% RSLogix 500 project High Pressure Washer no labels Veracruz.RSS, saved by version 11.00.00.00 %
PROJECT "UNTITLED"    % processor: MicroLogix 1400 %

PROGRAM FILES
  LAD 2   7 rungs
  LAD 3   25 rungs
  LAD 4   18 rungs
  LAD 5   20 rungs
  LAD 6   10 rungs
  LAD 7   39 rungs
  LAD 8   15 rungs
  LAD 9, 10, 11, 12, 13, 14, 15: only END

DATA FILES
  O0 OUTPUT  10 elements
  I1 INPUT  17 elements
  S2 STATUS  66 elements
  B3 BINARY  32 elements
  T4 TIMER  40 elements
  C5 COUNTER  32 elements
  R6 CONTROL  16 elements
  N7 INTEGER  110 elements
  F8 RESERVED  1 elements
  PD9   4 elements

LADDER 2
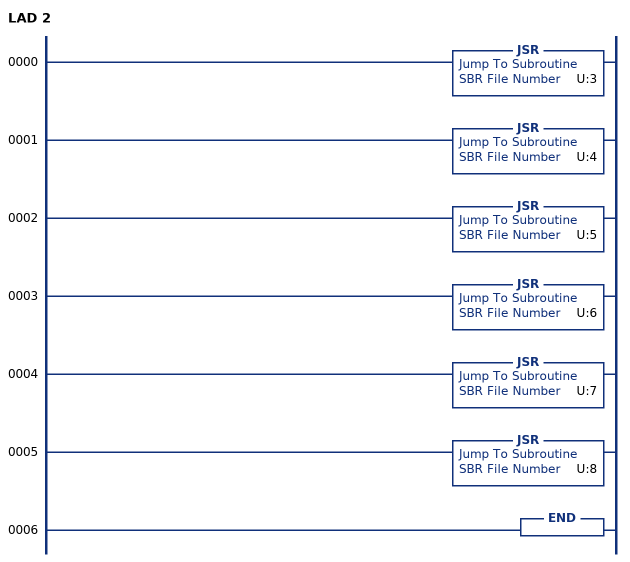
% Rung: 0 %
SOR JSR U:3 EOR
% Rung: 1 %
SOR JSR U:4 EOR
% Rung: 2 %
SOR JSR U:5 EOR
% Rung: 3 %
SOR JSR U:6 EOR
% Rung: 4 %
SOR JSR U:7 EOR
% Rung: 5 %
SOR JSR U:8 EOR
% Rung: 6 %
SOR END EOR

LADDER 3
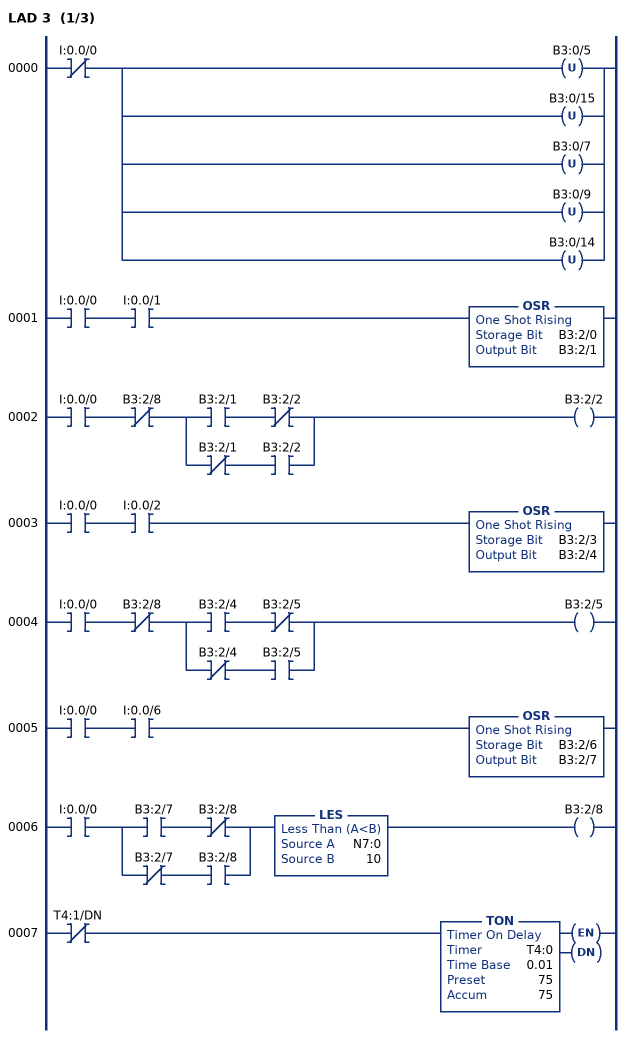
% Rung: 0 %
SOR XIO I:0.0/0 BST BST BST BST OTU B3:0/5 NXB OTU B3:0/15 BND NXB OTU B3:0/7 BND NXB OTU B3:0/9 BND NXB OTU B3:0/14 BND EOR
% Rung: 1 %
SOR XIC I:0.0/0 XIC I:0.0/1 OSR B3:2/0 B3:2/1 EOR
% Rung: 2 %
SOR XIC I:0.0/0 XIO B3:2/8 BST XIC B3:2/1 XIO B3:2/2 NXB XIO B3:2/1 XIC B3:2/2 BND OTE B3:2/2 EOR
% Rung: 3 %
SOR XIC I:0.0/0 XIC I:0.0/2 OSR B3:2/3 B3:2/4 EOR
% Rung: 4 %
SOR XIC I:0.0/0 XIO B3:2/8 BST XIC B3:2/4 XIO B3:2/5 NXB XIO B3:2/4 XIC B3:2/5 BND OTE B3:2/5 EOR
% Rung: 5 %
SOR XIC I:0.0/0 XIC I:0.0/6 OSR B3:2/6 B3:2/7 EOR
% Rung: 6 %
SOR XIC I:0.0/0 BST XIC B3:2/7 XIO B3:2/8 NXB XIO B3:2/7 XIC B3:2/8 BND LES N7:0 10 OTE B3:2/8 EOR
% Rung: 7 %
SOR XIO T4:1/DN TON T4:0 0.01 75 75 EOR

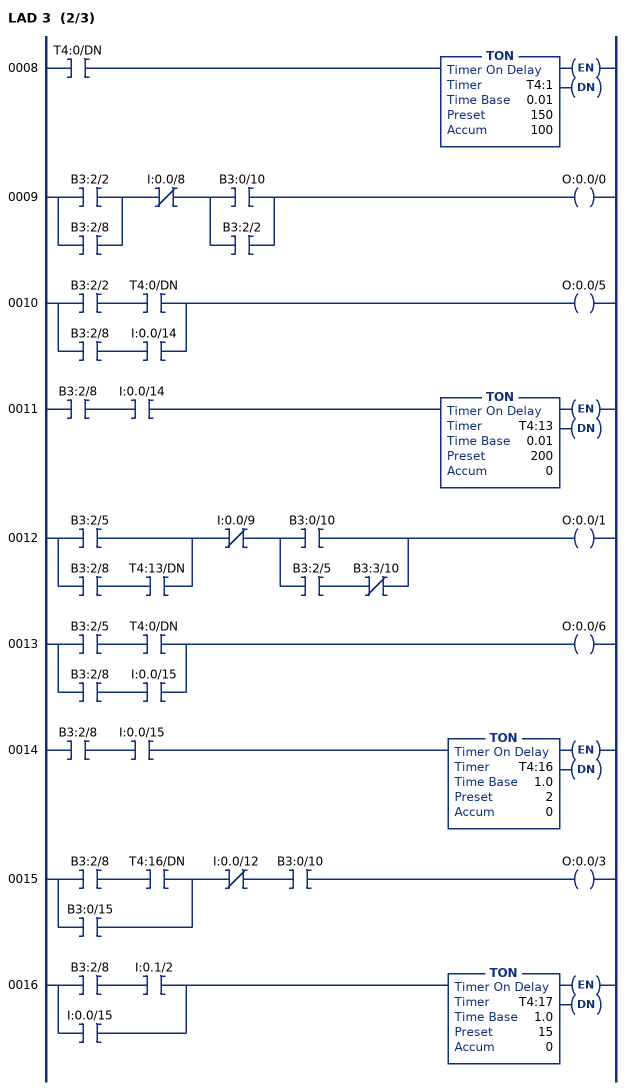
% Rung: 8 %
SOR XIC T4:0/DN TON T4:1 0.01 150 100 EOR
% Rung: 9 %
SOR BST XIC B3:2/2 NXB XIC B3:2/8 BND XIO I:0.0/8 BST XIC B3:0/10 NXB XIC B3:2/2 BND OTE O:0.0/0 EOR
% Rung: 10 %
SOR BST XIC B3:2/2 XIC T4:0/DN NXB XIC B3:2/8 XIC I:0.0/14 BND OTE O:0.0/5 EOR
% Rung: 11 %
SOR XIC B3:2/8 XIC I:0.0/14 TON T4:13 0.01 200 0 EOR
% Rung: 12 %
SOR BST XIC B3:2/5 NXB XIC B3:2/8 XIC T4:13/DN BND XIO I:0.0/9 BST XIC B3:0/10 NXB XIC B3:2/5 XIO B3:3/10 BND OTE O:0.0/1 EOR
% Rung: 13 %
SOR BST XIC B3:2/5 XIC T4:0/DN NXB XIC B3:2/8 XIC I:0.0/15 BND OTE O:0.0/6 EOR
% Rung: 14 %
SOR XIC B3:2/8 XIC I:0.0/15 TON T4:16 1.0 2 0 EOR
% Rung: 15 %
SOR BST XIC B3:2/8 XIC T4:16/DN NXB XIC B3:0/15 BND XIO I:0.0/12 XIC B3:0/10 OTE O:0.0/3 EOR
% Rung: 16 %
SOR BST XIC B3:2/8 XIC I:0.1/2 NXB XIC I:0.0/15 BND TON T4:17 1.0 15 0 EOR

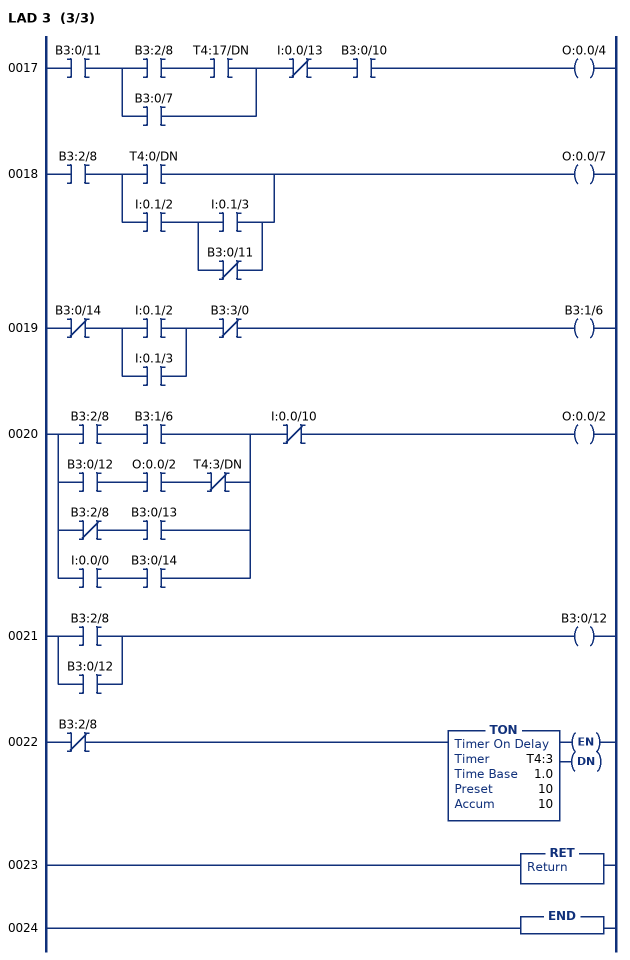
% Rung: 17 %
SOR XIC B3:0/11 BST XIC B3:2/8 XIC T4:17/DN NXB XIC B3:0/7 BND XIO I:0.0/13 XIC B3:0/10 OTE O:0.0/4 EOR
% Rung: 18 %
SOR XIC B3:2/8 BST XIC T4:0/DN NXB XIC I:0.1/2 BST XIC I:0.1/3 NXB XIO B3:0/11 BND BND OTE O:0.0/7 EOR
% Rung: 19 %
SOR XIO B3:0/14 BST XIC I:0.1/2 NXB XIC I:0.1/3 BND XIO B3:3/0 OTE B3:1/6 EOR
% Rung: 20 %
SOR BST BST BST XIC B3:2/8 XIC B3:1/6 NXB XIC B3:0/12 XIC O:0.0/2 XIO T4:3/DN BND NXB XIO B3:2/8 XIC B3:0/13 BND NXB XIC I:0.0/0 XIC B3:0/14 BND XIO I:0.0/10 OTE O:0.0/2 EOR
% Rung: 21 %
SOR BST XIC B3:2/8 NXB XIC B3:0/12 BND OTE B3:0/12 EOR
% Rung: 22 %
SOR XIO B3:2/8 TON T4:3 1.0 10 10 EOR
% Rung: 23 %
SOR RET EOR
% Rung: 24 %
SOR END EOR

LADDER 4
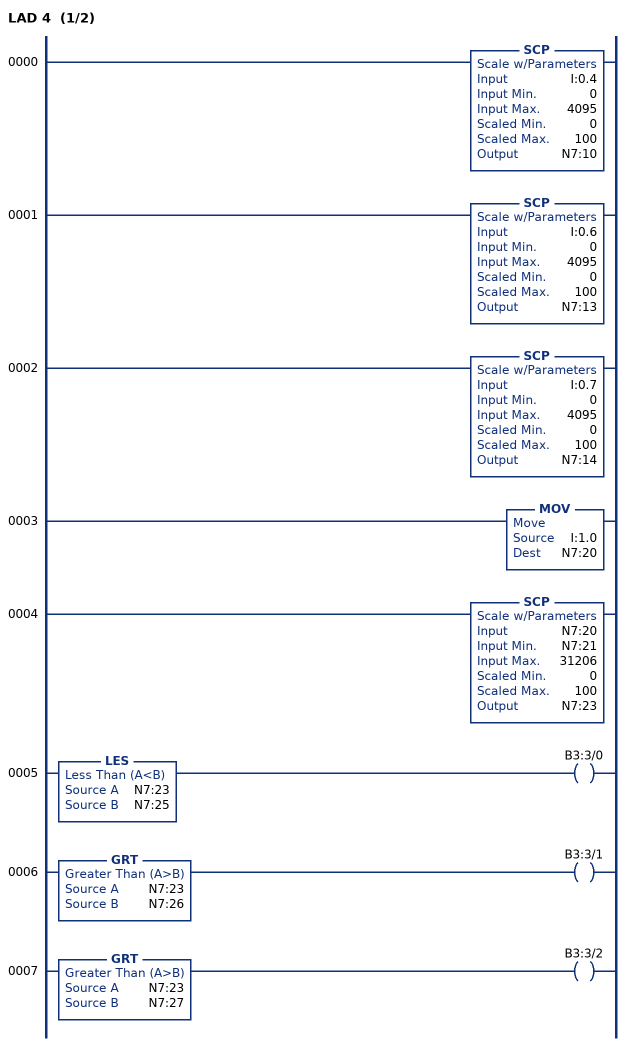
% Rung: 0 %
SOR SCP I:0.4 0 4095 0 100 N7:10 EOR
% Rung: 1 %
SOR SCP I:0.6 0 4095 0 100 N7:13 EOR
% Rung: 2 %
SOR SCP I:0.7 0 4095 0 100 N7:14 EOR
% Rung: 3 %
SOR MOV I:1.0 N7:20 EOR
% Rung: 4 %
SOR SCP N7:20 N7:21 31206 0 100 N7:23 EOR
% Rung: 5 %
SOR LES N7:23 N7:25 OTE B3:3/0 EOR
% Rung: 6 %
SOR GRT N7:23 N7:26 OTE B3:3/1 EOR
% Rung: 7 %
SOR GRT N7:23 N7:27 OTE B3:3/2 EOR

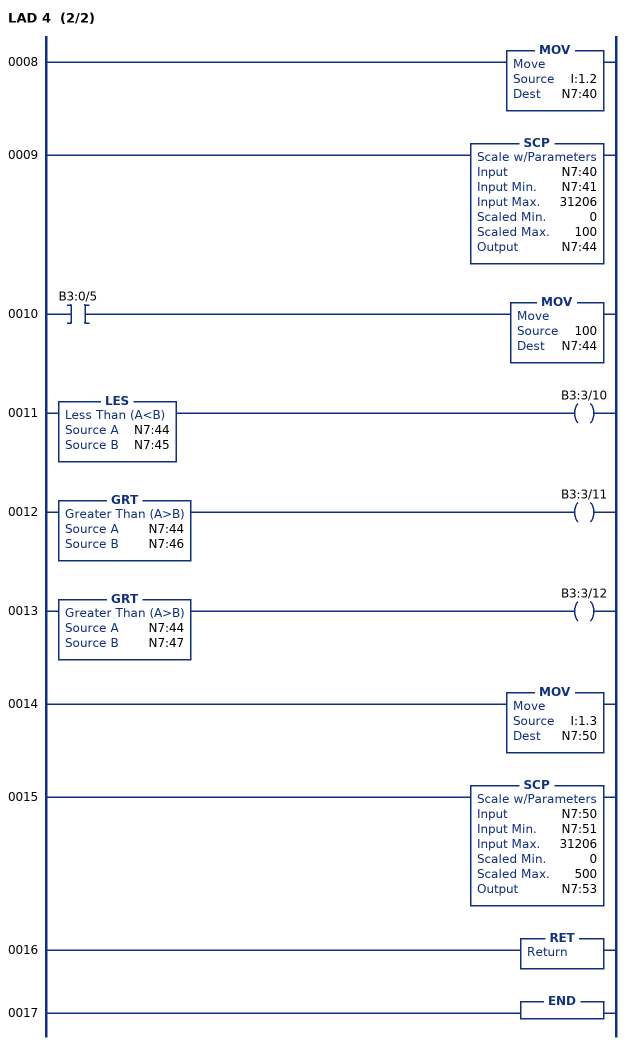
% Rung: 8 %
SOR MOV I:1.2 N7:40 EOR
% Rung: 9 %
SOR SCP N7:40 N7:41 31206 0 100 N7:44 EOR
% Rung: 10 %
SOR XIC B3:0/5 MOV 100 N7:44 EOR
% Rung: 11 %
SOR LES N7:44 N7:45 OTE B3:3/10 EOR
% Rung: 12 %
SOR GRT N7:44 N7:46 OTE B3:3/11 EOR
% Rung: 13 %
SOR GRT N7:44 N7:47 OTE B3:3/12 EOR
% Rung: 14 %
SOR MOV I:1.3 N7:50 EOR
% Rung: 15 %
SOR SCP N7:50 N7:51 31206 0 500 N7:53 EOR
% Rung: 16 %
SOR RET EOR
% Rung: 17 %
SOR END EOR

LADDER 5
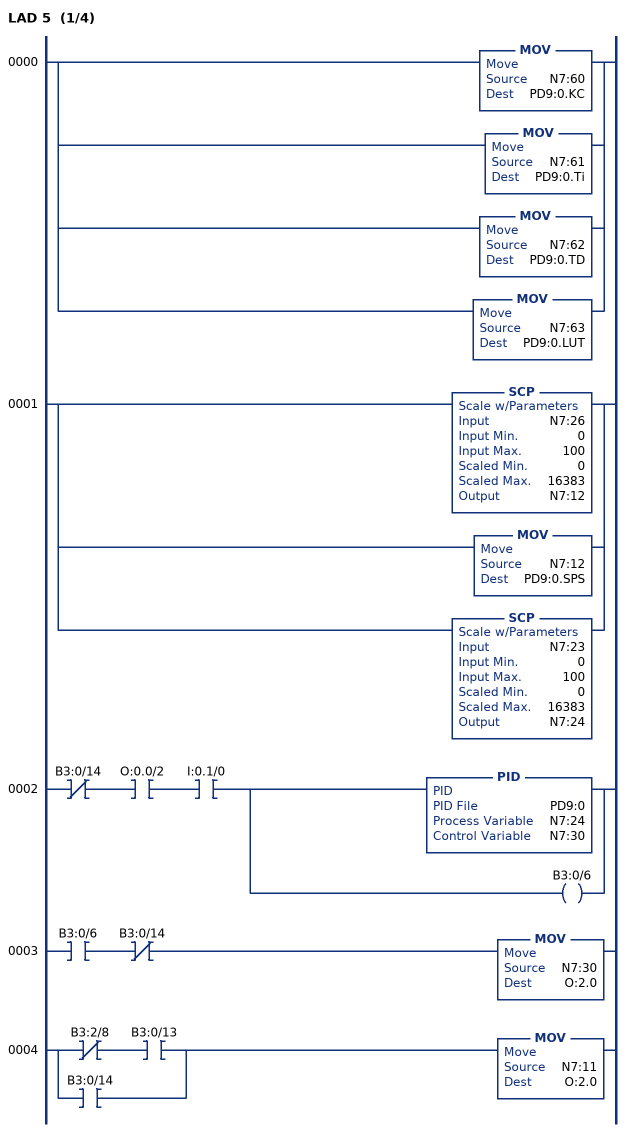
% Rung: 0 %
SOR BST BST BST MOV N7:60 PD9:0.KC NXB MOV N7:61 PD9:0.Ti BND NXB MOV N7:62 PD9:0.TD BND NXB MOV N7:63 PD9:0.LUT BND EOR
% Rung: 1 %
SOR BST SCP N7:26 0 100 0 16383 N7:12 NXB BST MOV N7:12 PD9:0.SPS NXB SCP N7:23 0 100 0 16383 N7:24 BND BND EOR
% Rung: 2 %
SOR XIO B3:0/14 XIC O:0.0/2 XIC I:0.1/0 BST PID PD9:0 N7:24 N7:30 NXB OTE B3:0/6 BND EOR
% Rung: 3 %
SOR XIC B3:0/6 XIO B3:0/14 MOV N7:30 O:2.0 EOR
% Rung: 4 %
SOR BST XIO B3:2/8 XIC B3:0/13 NXB XIC B3:0/14 BND MOV N7:11 O:2.0 EOR

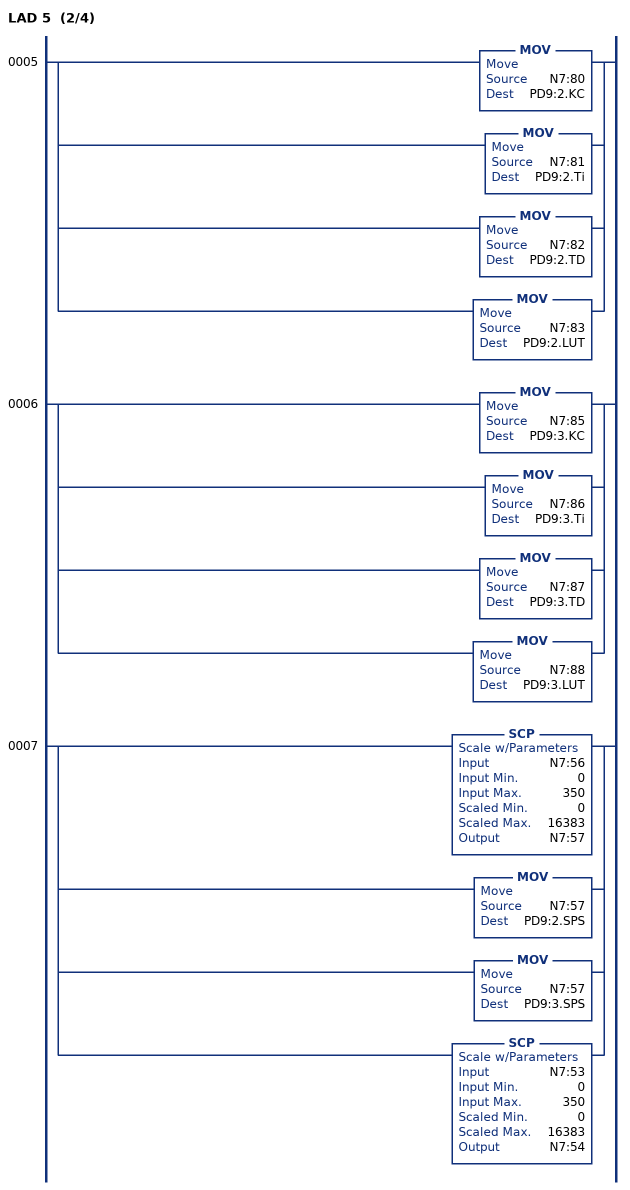
% Rung: 5 %
SOR BST BST BST MOV N7:80 PD9:2.KC NXB MOV N7:81 PD9:2.Ti BND NXB MOV N7:82 PD9:2.TD BND NXB MOV N7:83 PD9:2.LUT BND EOR
% Rung: 6 %
SOR BST BST BST MOV N7:85 PD9:3.KC NXB MOV N7:86 PD9:3.Ti BND NXB MOV N7:87 PD9:3.TD BND NXB MOV N7:88 PD9:3.LUT BND EOR
% Rung: 7 %
SOR BST SCP N7:56 0 350 0 16383 N7:57 NXB BST BST MOV N7:57 PD9:2.SPS NXB MOV N7:57 PD9:3.SPS BND NXB SCP N7:53 0 350 0 16383 N7:54 BND BND EOR

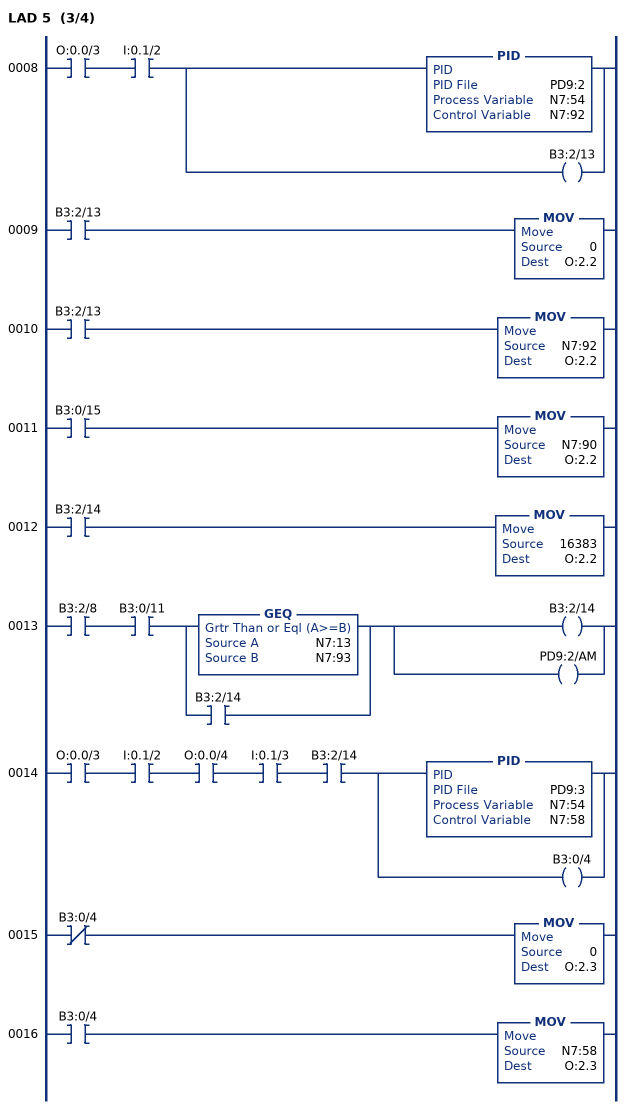
% Rung: 8 %
SOR XIC O:0.0/3 XIC I:0.1/2 BST PID PD9:2 N7:54 N7:92 NXB OTE B3:2/13 BND EOR
% Rung: 9 %
SOR XIC B3:2/13 MOV 0 O:2.2 EOR
% Rung: 10 %
SOR XIC B3:2/13 MOV N7:92 O:2.2 EOR
% Rung: 11 %
SOR XIC B3:0/15 MOV N7:90 O:2.2 EOR
% Rung: 12 %
SOR XIC B3:2/14 MOV 16383 O:2.2 EOR
% Rung: 13 %
SOR XIC B3:2/8 XIC B3:0/11 BST GEQ N7:13 N7:93 NXB XIC B3:2/14 BND BST OTE B3:2/14 NXB OTE PD9:2/AM BND EOR
% Rung: 14 %
SOR XIC O:0.0/3 XIC I:0.1/2 XIC O:0.0/4 XIC I:0.1/3 XIC B3:2/14 BST PID PD9:3 N7:54 N7:58 NXB OTE B3:0/4 BND EOR
% Rung: 15 %
SOR XIO B3:0/4 MOV 0 O:2.3 EOR
% Rung: 16 %
SOR XIC B3:0/4 MOV N7:58 O:2.3 EOR

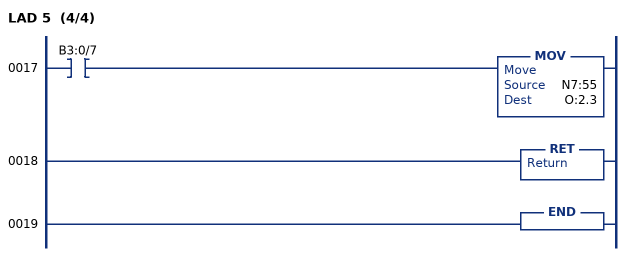
% Rung: 17 %
SOR XIC B3:0/7 MOV N7:55 O:2.3 EOR
% Rung: 18 %
SOR RET EOR
% Rung: 19 %
SOR END EOR

LADDER 6
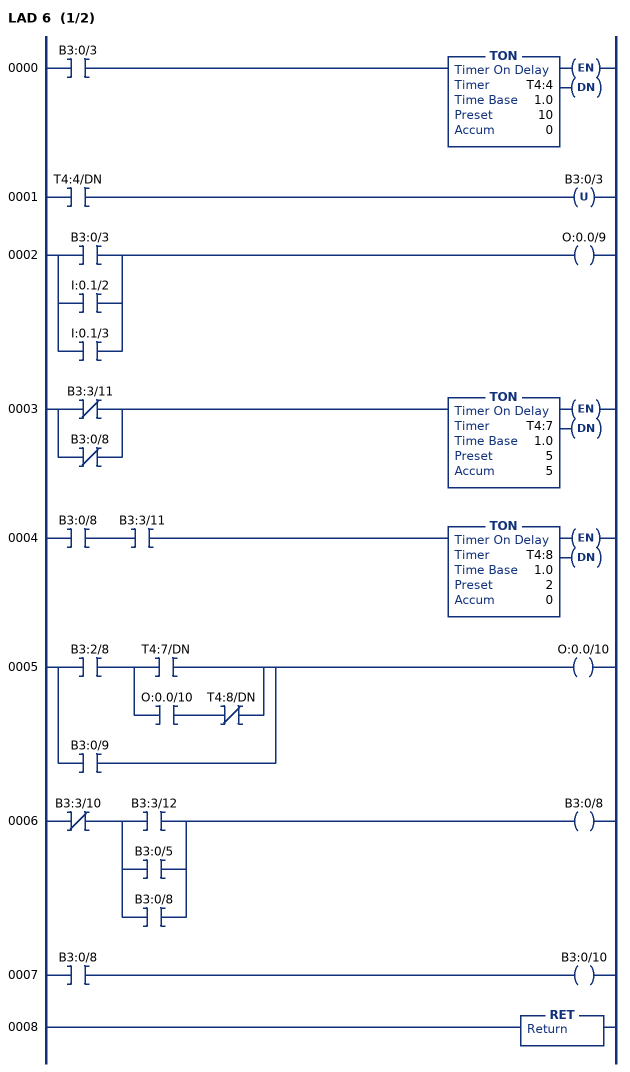
% Rung: 0 %
SOR XIC B3:0/3 TON T4:4 1.0 10 0 EOR
% Rung: 1 %
SOR XIC T4:4/DN OTU B3:0/3 EOR
% Rung: 2 %
SOR BST BST XIC B3:0/3 NXB XIC I:0.1/2 BND NXB XIC I:0.1/3 BND OTE O:0.0/9 EOR
% Rung: 3 %
SOR BST XIO B3:3/11 NXB XIO B3:0/8 BND TON T4:7 1.0 5 5 EOR
% Rung: 4 %
SOR XIC B3:0/8 XIC B3:3/11 TON T4:8 1.0 2 0 EOR
% Rung: 5 %
SOR BST XIC B3:2/8 BST XIC T4:7/DN NXB XIC O:0.0/10 XIO T4:8/DN BND NXB XIC B3:0/9 BND OTE O:0.0/10 EOR
% Rung: 6 %
SOR XIO B3:3/10 BST BST XIC B3:3/12 NXB XIC B3:0/5 BND NXB XIC B3:0/8 BND OTE B3:0/8 EOR
% Rung: 7 %
SOR XIC B3:0/8 OTE B3:0/10 EOR
% Rung: 8 %
SOR RET EOR

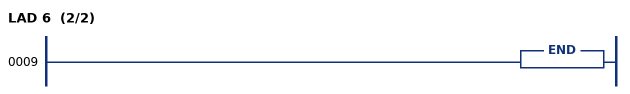
% Rung: 9 %
SOR END EOR

LADDER 7
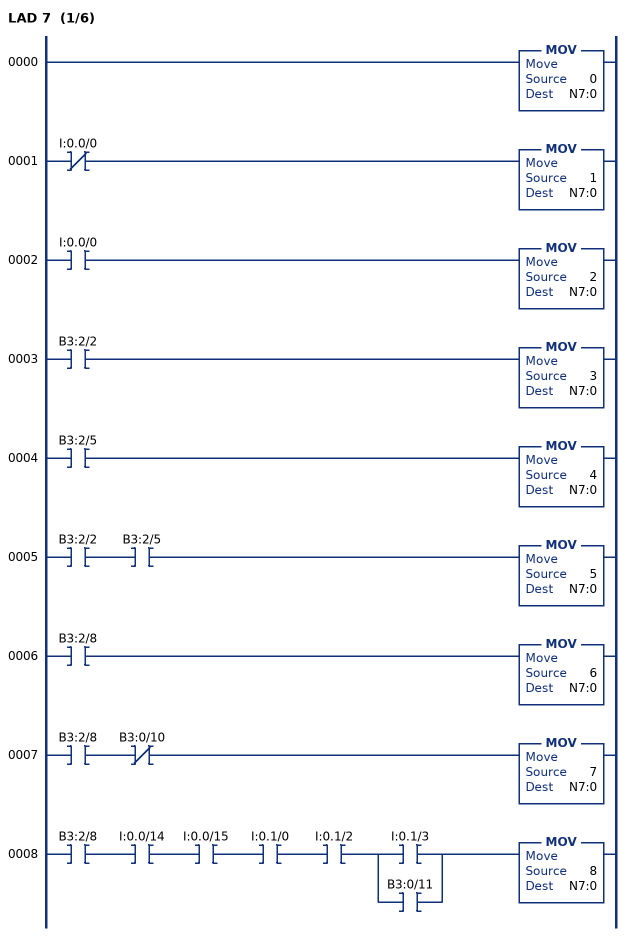
% Rung: 0 %
SOR MOV 0 N7:0 EOR
% Rung: 1 %
SOR XIO I:0.0/0 MOV 1 N7:0 EOR
% Rung: 2 %
SOR XIC I:0.0/0 MOV 2 N7:0 EOR
% Rung: 3 %
SOR XIC B3:2/2 MOV 3 N7:0 EOR
% Rung: 4 %
SOR XIC B3:2/5 MOV 4 N7:0 EOR
% Rung: 5 %
SOR XIC B3:2/2 XIC B3:2/5 MOV 5 N7:0 EOR
% Rung: 6 %
SOR XIC B3:2/8 MOV 6 N7:0 EOR
% Rung: 7 %
SOR XIC B3:2/8 XIO B3:0/10 MOV 7 N7:0 EOR
% Rung: 8 %
SOR XIC B3:2/8 XIC I:0.0/14 XIC I:0.0/15 XIC I:0.1/0 XIC I:0.1/2 BST XIC I:0.1/3 NXB XIC B3:0/11 BND MOV 8 N7:0 EOR

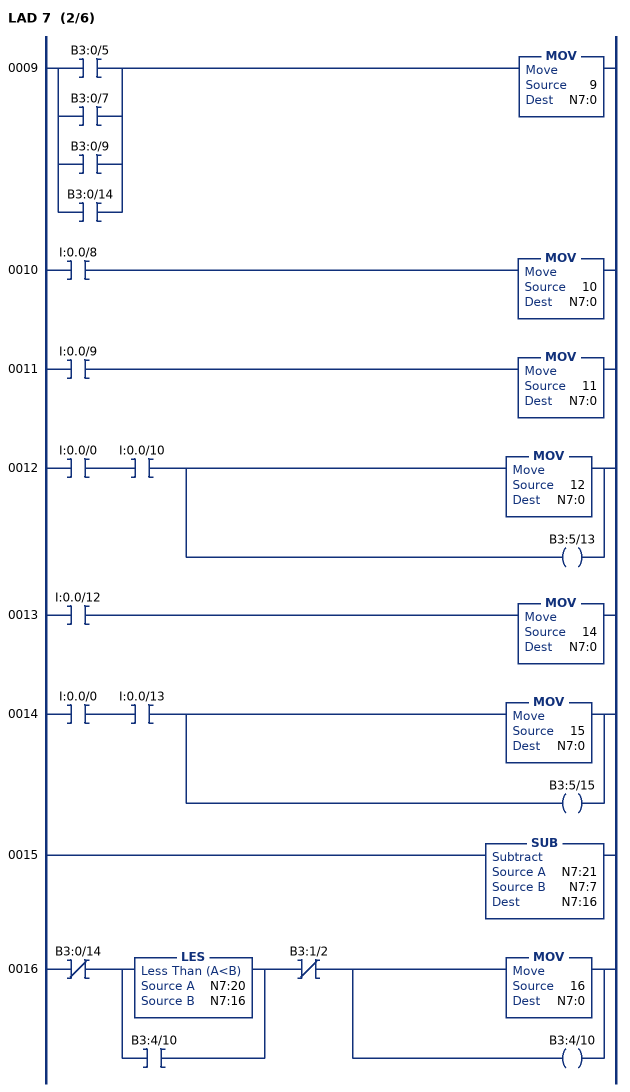
% Rung: 9 %
SOR BST BST BST XIC B3:0/5 NXB XIC B3:0/7 BND NXB XIC B3:0/9 BND NXB XIC B3:0/14 BND MOV 9 N7:0 EOR
% Rung: 10 %
SOR XIC I:0.0/8 MOV 10 N7:0 EOR
% Rung: 11 %
SOR XIC I:0.0/9 MOV 11 N7:0 EOR
% Rung: 12 %
SOR XIC I:0.0/0 XIC I:0.0/10 BST MOV 12 N7:0 NXB OTE B3:5/13 BND EOR
% Rung: 13 %
SOR XIC I:0.0/12 MOV 14 N7:0 EOR
% Rung: 14 %
SOR XIC I:0.0/0 XIC I:0.0/13 BST MOV 15 N7:0 NXB OTE B3:5/15 BND EOR
% Rung: 15 %
SOR SUB N7:21 N7:7 N7:16 EOR
% Rung: 16 %
SOR XIO B3:0/14 BST LES N7:20 N7:16 NXB XIC B3:4/10 BND XIO B3:1/2 BST MOV 16 N7:0 NXB OTE B3:4/10 BND EOR

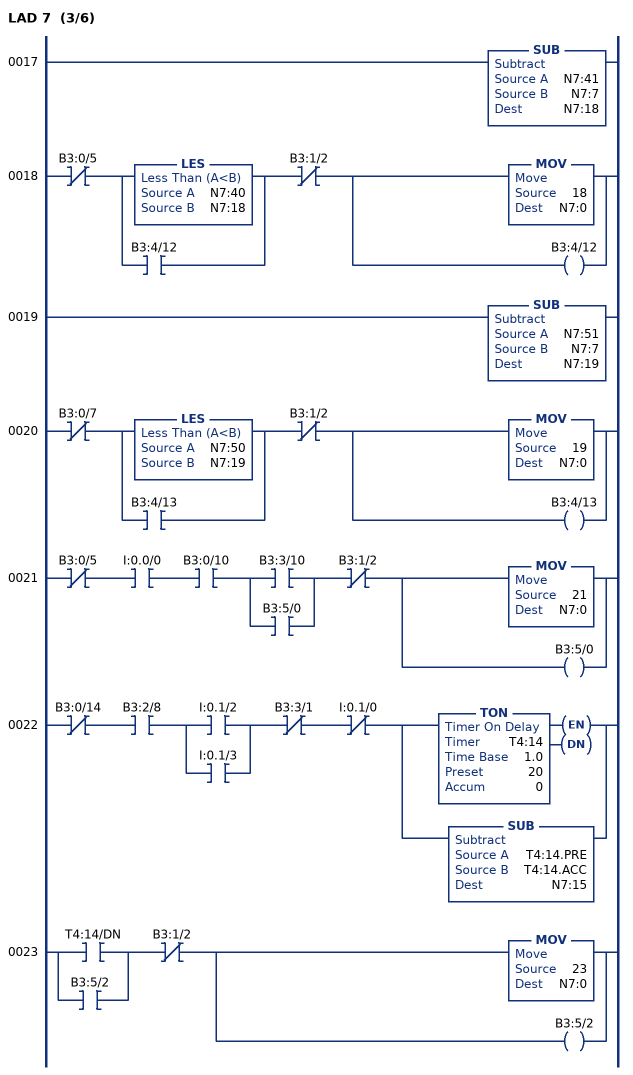
% Rung: 17 %
SOR SUB N7:41 N7:7 N7:18 EOR
% Rung: 18 %
SOR XIO B3:0/5 BST LES N7:40 N7:18 NXB XIC B3:4/12 BND XIO B3:1/2 BST MOV 18 N7:0 NXB OTE B3:4/12 BND EOR
% Rung: 19 %
SOR SUB N7:51 N7:7 N7:19 EOR
% Rung: 20 %
SOR XIO B3:0/7 BST LES N7:50 N7:19 NXB XIC B3:4/13 BND XIO B3:1/2 BST MOV 19 N7:0 NXB OTE B3:4/13 BND EOR
% Rung: 21 %
SOR XIO B3:0/5 XIC I:0.0/0 XIC B3:0/10 BST XIC B3:3/10 NXB XIC B3:5/0 BND XIO B3:1/2 BST MOV 21 N7:0 NXB OTE B3:5/0 BND EOR
% Rung: 22 %
SOR XIO B3:0/14 XIC B3:2/8 BST XIC I:0.1/2 NXB XIC I:0.1/3 BND XIO B3:3/1 XIO I:0.1/0 BST TON T4:14 1.0 20 0 NXB SUB T4:14.PRE T4:14.ACC N7:15 BND EOR
% Rung: 23 %
SOR BST XIC T4:14/DN NXB XIC B3:5/2 BND XIO B3:1/2 BST MOV 23 N7:0 NXB OTE B3:5/2 BND EOR

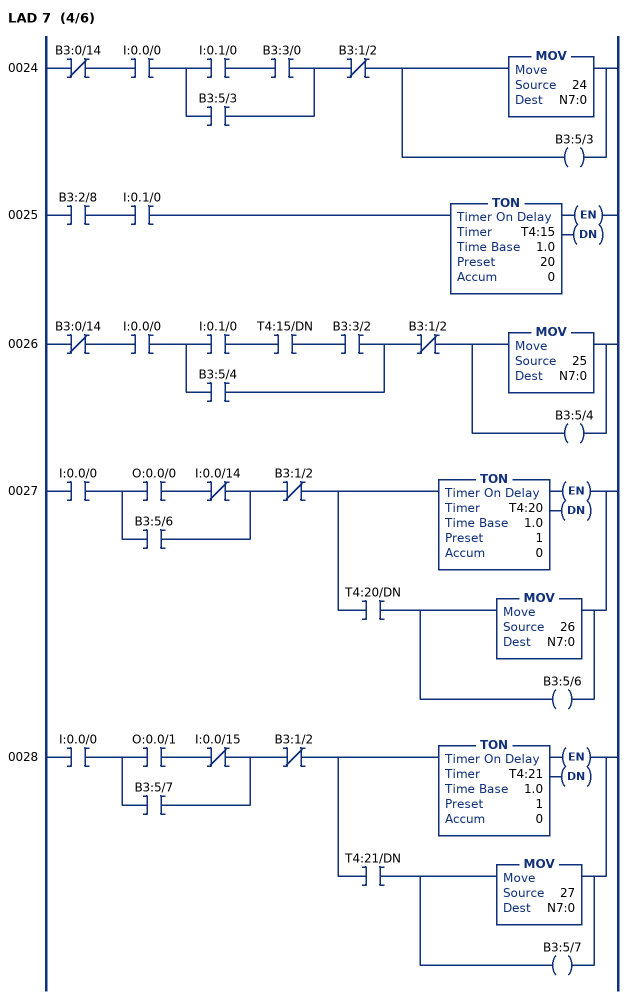
% Rung: 24 %
SOR XIO B3:0/14 XIC I:0.0/0 BST XIC I:0.1/0 XIC B3:3/0 NXB XIC B3:5/3 BND XIO B3:1/2 BST MOV 24 N7:0 NXB OTE B3:5/3 BND EOR
% Rung: 25 %
SOR XIC B3:2/8 XIC I:0.1/0 TON T4:15 1.0 20 0 EOR
% Rung: 26 %
SOR XIO B3:0/14 XIC I:0.0/0 BST XIC I:0.1/0 XIC T4:15/DN XIC B3:3/2 NXB XIC B3:5/4 BND XIO B3:1/2 BST MOV 25 N7:0 NXB OTE B3:5/4 BND EOR
% Rung: 27 %
SOR XIC I:0.0/0 BST XIC O:0.0/0 XIO I:0.0/14 NXB XIC B3:5/6 BND XIO B3:1/2 BST TON T4:20 1.0 1 0 NXB XIC T4:20/DN BST MOV 26 N7:0 NXB OTE B3:5/6 BND BND EOR
% Rung: 28 %
SOR XIC I:0.0/0 BST XIC O:0.0/1 XIO I:0.0/15 NXB XIC B3:5/7 BND XIO B3:1/2 BST TON T4:21 1.0 1 0 NXB XIC T4:21/DN BST MOV 27 N7:0 NXB OTE B3:5/7 BND BND EOR

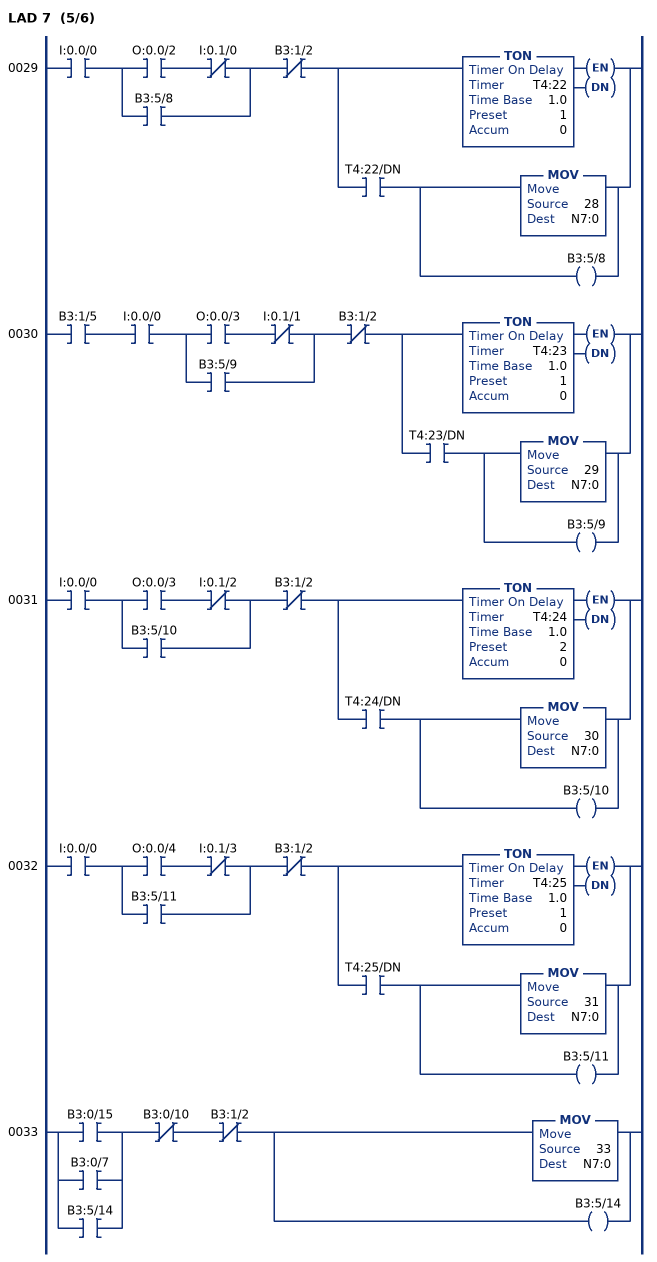
% Rung: 29 %
SOR XIC I:0.0/0 BST XIC O:0.0/2 XIO I:0.1/0 NXB XIC B3:5/8 BND XIO B3:1/2 BST TON T4:22 1.0 1 0 NXB XIC T4:22/DN BST MOV 28 N7:0 NXB OTE B3:5/8 BND BND EOR
% Rung: 30 %
SOR XIC B3:1/5 XIC I:0.0/0 BST XIC O:0.0/3 XIO I:0.1/1 NXB XIC B3:5/9 BND XIO B3:1/2 BST TON T4:23 1.0 1 0 NXB XIC T4:23/DN BST MOV 29 N7:0 NXB OTE B3:5/9 BND BND EOR
% Rung: 31 %
SOR XIC I:0.0/0 BST XIC O:0.0/3 XIO I:0.1/2 NXB XIC B3:5/10 BND XIO B3:1/2 BST TON T4:24 1.0 2 0 NXB XIC T4:24/DN BST MOV 30 N7:0 NXB OTE B3:5/10 BND BND EOR
% Rung: 32 %
SOR XIC I:0.0/0 BST XIC O:0.0/4 XIO I:0.1/3 NXB XIC B3:5/11 BND XIO B3:1/2 BST TON T4:25 1.0 1 0 NXB XIC T4:25/DN BST MOV 31 N7:0 NXB OTE B3:5/11 BND BND EOR
% Rung: 33 %
SOR BST BST XIC B3:0/15 NXB XIC B3:0/7 BND NXB XIC B3:5/14 BND XIO B3:0/10 XIO B3:1/2 BST MOV 33 N7:0 NXB OTE B3:5/14 BND EOR

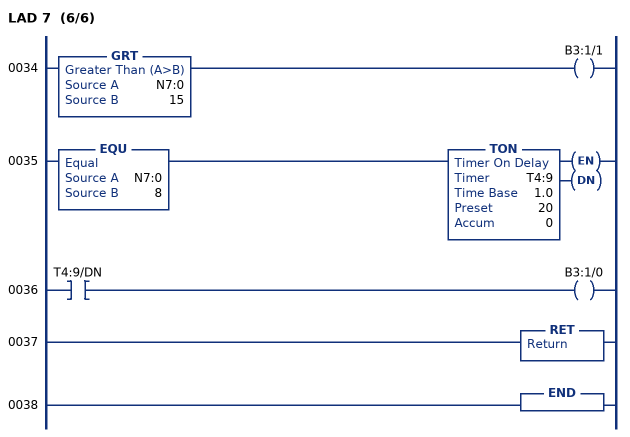
% Rung: 34 %
SOR GRT N7:0 15 OTE B3:1/1 EOR
% Rung: 35 %
SOR EQU N7:0 8 TON T4:9 1.0 20 0 EOR
% Rung: 36 %
SOR XIC T4:9/DN OTE B3:1/0 EOR
% Rung: 37 %
SOR RET EOR
% Rung: 38 %
SOR END EOR

LADDER 8
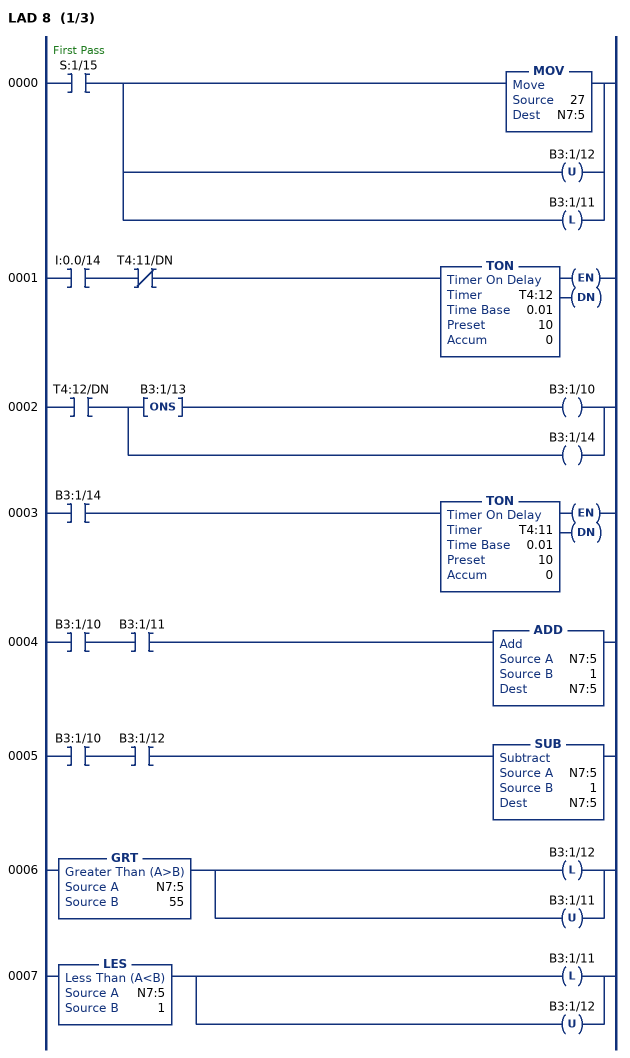
% Rung: 0 %
SOR XIC S:1/15 BST MOV 27 N7:5 NXB BST OTU B3:1/12 NXB OTL B3:1/11 BND BND EOR
%   S:1/15  "First Pass" %
% Rung: 1 %
SOR XIC I:0.0/14 XIO T4:11/DN TON T4:12 0.01 10 0 EOR
% Rung: 2 %
SOR XIC T4:12/DN BST ONS B3:1/13 OTE B3:1/10 NXB OTE B3:1/14 BND EOR
% Rung: 3 %
SOR XIC B3:1/14 TON T4:11 0.01 10 0 EOR
% Rung: 4 %
SOR XIC B3:1/10 XIC B3:1/11 ADD N7:5 1 N7:5 EOR
% Rung: 5 %
SOR XIC B3:1/10 XIC B3:1/12 SUB N7:5 1 N7:5 EOR
% Rung: 6 %
SOR GRT N7:5 55 BST OTL B3:1/12 NXB OTU B3:1/11 BND EOR
% Rung: 7 %
SOR LES N7:5 1 BST OTL B3:1/11 NXB OTU B3:1/12 BND EOR

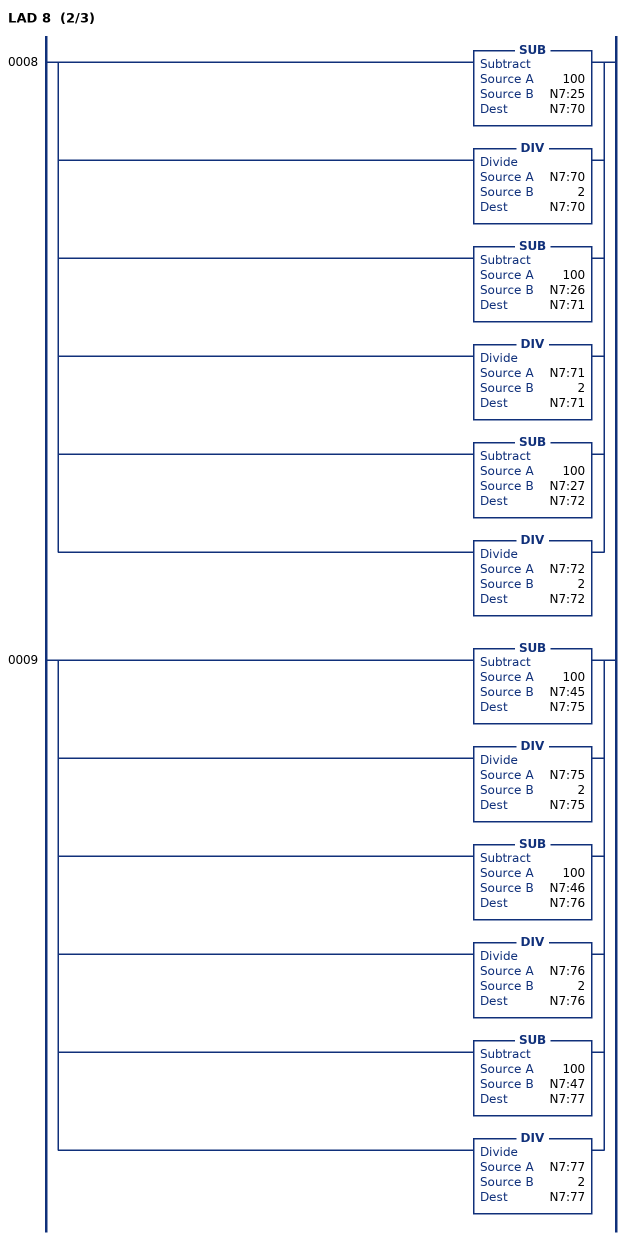
% Rung: 8 %
SOR BST BST SUB 100 N7:25 N7:70 NXB DIV N7:70 2 N7:70 BND NXB BST BST SUB 100 N7:26 N7:71 NXB DIV N7:71 2 N7:71 BND NXB BST SUB 100 N7:27 N7:72 NXB DIV N7:72 2 N7:72 BND BND BND EOR
% Rung: 9 %
SOR BST BST SUB 100 N7:45 N7:75 NXB DIV N7:75 2 N7:75 BND NXB BST BST SUB 100 N7:46 N7:76 NXB DIV N7:76 2 N7:76 BND NXB BST SUB 100 N7:47 N7:77 NXB DIV N7:77 2 N7:77 BND BND BND EOR

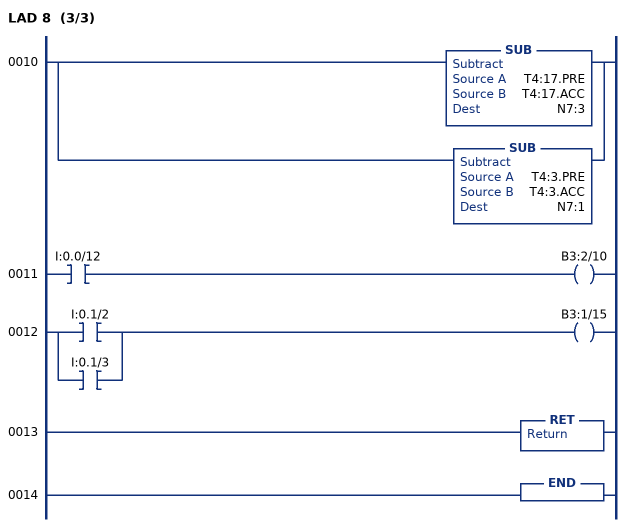
% Rung: 10 %
SOR BST SUB T4:17.PRE T4:17.ACC N7:3 NXB SUB T4:3.PRE T4:3.ACC N7:1 BND EOR
% Rung: 11 %
SOR XIC I:0.0/12 OTE B3:2/10 EOR
% Rung: 12 %
SOR BST XIC I:0.1/2 NXB XIC I:0.1/3 BND OTE B3:1/15 EOR
% Rung: 13 %
SOR RET EOR
% Rung: 14 %
SOR END EOR

DATA TABLE (non-zero values as saved)
DATA B3
% B3:0 % 0X1500 0X0800 0X0000 0X0002 0X0000 0X0000 0X0000 0X0000 0X0000 0X0000
DATA T4
% .PRE .ACC %
% T4:0 % 75 75
% T4:1 % 150 100
% T4:2 % 2 0
% T4:3 % 10 10
% T4:4 % 10 0
% T4:5 % 10 0
% T4:6 % 50 0
% T4:7 % 5 5
% T4:8 % 2 0
% T4:9 % 20 0
% T4:10 % 2 0
% T4:11 % 10 0
% T4:12 % 10 0
% T4:13 % 200 0
% T4:14 % 20 0
% T4:15 % 20 0
% T4:16 % 2 0
% T4:17 % 15 0
% T4:20 % 1 0
% T4:21 % 1 0
% T4:22 % 1 0
% T4:23 % 1 0
% T4:24 % 2 0
% T4:25 % 1 0
DATA C5
% .PRE .ACC %
% C5:0 % 1000 7
% C5:1 % 27 1
DATA N7
% N7:0 % 2 0 0 15 0 40 0 20 0 0
% N7:10 % 0 6553 4915 0 0 14 6230 0 6230 6410
% N7:20 % 19811 6250 100 54 8847 18 30 55 0 0
% N7:30 % 3747 0 0 0 0 0 0 0 0 16383
% N7:40 % 19829 6250 100 0 54 20 80 100 0 0
% N7:50 % 6441 6430 500 0 0 0 35 1638 3103 0
% N7:60 % 10 5 0 300 0 10 5 0 50 0
% N7:70 % 41 35 23 0 0 40 10 0 0 0
% N7:80 % 40 1 0 50 0 10 5 0 300 0
% N7:90 % 0 0 10134 100 90 0 0 0 0 0
